PROGRAM Alarm_conv_3
VAR
bAlarm_b3_S1_SB0_blink	:BOOL;
bAlarm_b3_S6_SB0_blink	:BOOL;
END_VAR

//Нет готовности конвейер 3	
	bAlarm3QF2_3QF7 S=NOT b_3QF2_3QF7 	AND bPermAlarm1;
	bAlarm3QF8 		S=NOT b_3QF8 		AND bPermAlarm1;
//	bAlarm3KM2 		S=NOT b_3KM2 		AND bPermAlarm1;
//	bAlarm3KM3 		S=NOT b_3KM3 		AND bPermAlarm1;
//	bAlarm3KM4 		S=NOT b_3KM4 		AND bPermAlarm1;
//	bAlarm3KM5 		S=NOT b_3KM5 		AND bPermAlarm1;
//	bAlarm3KM6 		S=NOT b_3KM6 		AND bPermAlarm1;
//	bAlarm3KM7 		S=NOT b_3KM7 		AND bPermAlarm1;
	
//Грибки
	bAlarm_b3_S1_SB0 S=NOT   b3_S1_SB0 	AND bPermAlarm1;
	bAlarm_b3_S6_SB0 S=NOT   b3_S6_SB0 	AND bPermAlarm1;

// Индикация на грибках
	b3S1_SB0 := NOT b3_S1_SB0 AND blink.OUT;
	b3S6_SB0 := NOT b3_S6_SB0 AND blink.OUT;	
	
	blink(ENABLE:=bAlarm_b3_S1_SB0,TIMELOW:=T#500MS,TIMEHIGH:=T#500MS);
	bAlarm_b3_S1_SB0_blink := blink.OUT AND bAlarm_b3_S1_SB0;
	bAlarm_b3_S6_SB0_blink := blink.OUT AND bAlarm_b3_S6_SB0;	
(*Авария безопасности*)
	bAlarmSafety3 := bAlarm_b3_S1_SB0 OR bAlarm_b3_S6_SB0;

(*Нет общей готовности конвейера 1*)
	bNotReady_3 := bAlarm3QF2_3QF7 OR bAlarm3QF8 OR bAlarm3KM2 OR bAlarm3KM3 OR bAlarm3KM4 OR bAlarm3KM5 OR bAlarm3KM6 OR bAlarm3KM7;
					
IF  bNotReady3 THEN  sAlarm3:="Нет готовности 3";
		ELSIF bAlarmSafety3 THEN  sAlarm2:="Авария безопасности 3";
			ELSE sAlarm3:="---------";
END_IF

	bPermAlarmDrive3 := bPermAlarm1 AND NOT bAlarmSafety3;

(*(*Готовность *)
	IF NOT bDriveReady3s01M1 AND bPermAlarmDrive3  THEN  bNotDriveReady3s01M1 := TRUE;
	END_IF    
	IF NOT bDriveReady3s02M1 AND bPermAlarmDrive3  THEN  bNotDriveReady3s02M1 := TRUE;
	END_IF 
	IF NOT bDriveReady3s03M1 AND bPermAlarmDrive3  THEN  bNotDriveReady3s03M1 := TRUE;
	END_IF 
	IF NOT bDriveReady3s04M1 AND bPermAlarmDrive3  THEN  bNotDriveReady3s04M1 := TRUE;
	END_IF 
	IF NOT bDriveReady3s05M1 AND bPermAlarmDrive3  THEN  bNotDriveReady3s05M1 := TRUE;
	END_IF 
	IF NOT bDriveReady3s06M1 AND bPermAlarmDrive3  THEN  bNotDriveReady3s06M1 := TRUE;
	END_IF*)

(*Долгие перемещения Drive*)
	IF bLongMove3s01_s02_1   THEN bLongMove_3s01_s02_1 := TRUE;
	END_IF
	IF bLongMove3s02_1_s02_2  THEN bLongMove_3s02_1_s02_2 := TRUE;
	END_IF
	IF bLongMove3s02_2_s03_1  THEN bLongMove_3s02_2_s03_1 := TRUE;
	END_IF
	IF bLongMove3s02_s03  THEN bLongMove_3s02_s03 := TRUE;
	END_IF
		IF bLongMove3s03_1_s03_2   THEN bLongMove_3s03_1_s03_2 := TRUE;
	END_IF
	IF bLongMove3s03_2_s04_1  THEN bLongMove_3s03_2_s04_1 := TRUE;
	END_IF
	IF bLongMove3s03_s04  THEN bLongMove_3s03_s04 := TRUE;
	END_IF
	IF bLongMove3s04_1_s04_2  THEN bLongMove_3s04_1_s04_2 := TRUE;
	END_IF
		IF bLongMove3s04_2_s05   THEN bLongMove_3s04_2_s05  := TRUE;
	END_IF
	IF bLongMove3s05_1s06  THEN bLongMove_3s05_1s06 := TRUE;	
	END_IF
	
(*Нет готовности*)
	bNotReady3 := bNotDriveReady3s01M1 OR bNotDriveReady3s02M1 OR bNotDriveReady3s03M1 OR
			  bNotDriveReady3s04M1 OR bNotDriveReady3s05M1 OR bNotDriveReady3s06M1;

(*Долгое премещение*)
	bLongMove3 :=bLongMove_3s02_1_s02_2 OR bLongMove_3s02_1_s02_2  OR bLongMove_3s02_s03 OR
	       bLongMove_3s03_1_s03_2 OR bLongMove_3s03_2_s04_1 OR bLongMove_3s03_s04 OR bLongMove_3s04_1_s04_2 OR
			bLongMove_3s04_2_s05   OR bLongMove_3s05_1s06;


(*Сброс бита аварии по кнопке с панели*)
	bAlarmReset3 := bButtAlarmReset3;

(*Восстановление/сброс аварийных сигналов*)
IF bReset3 OR bAlarmReset3 THEN
	bAlarm3QF8 :=FALSE; bAlarm3QF2_3QF7 :=FALSE; 
	bAlarm3KM2 :=FALSE; bAlarm3KM3 :=FALSE; bAlarm3KM4 :=FALSE; bAlarm3KM5 :=FALSE; bAlarm3KM6 :=FALSE; bAlarm3KM7 :=FALSE;

	bNotDriveReady3s01M1 := FALSE; bNotDriveReady3s02M1 := FALSE; bNotDriveReady3s03M1 := FALSE;
	bNotDriveReady3s04M1 := FALSE; bNotDriveReady3s05M1 := FALSE; bNotDriveReady3s06M1 := FALSE;
	
	bLongMove_3s02_1_s02_2 := FALSE;bLongMove_3s02_1_s02_2 := FALSE; bLongMove_3s02_s03 := FALSE;
	bLongMove_3s03_1_s03_2 := FALSE; bLongMove_3s03_2_s04_1:= FALSE; bLongMove_3s03_s04 := FALSE;
	 bLongMove_3s04_1_s04_2:= FALSE;  bLongMove_3s04_2_s05 := FALSE;
    bLongMove_3s05_1s06 := FALSE;
	
	
	bAlarm_b3_S1_SB0 := FALSE; bAlarm_b3_S6_SB0 := FALSE;
END_IF

(*Формирование аварии*)
	bAlarm3 := bNotReady3 OR bLongMove3 OR bAlarmSafety3 OR bNotReady_3 OR bNotReadyGeneral OR bOverflow_CTU_Weight3 OR bOverflow_CTU_ID3;
	bAlarm3_vis := blink.OUT AND bAlarm3;
	
IF  bNotReady3 THEN  sAlarmLine3:="Нет готовности 3";
		ELSIF bLongMove3 THEN   sAlarmLine3:="Долгое перемещение 3";
			ELSE sAlarmLine3:="---------";
END_IF
IF bAlarm3 AND b_3AS1 THEN bRed_3S1HL1 :=TRUE; bRed_3S1_HL1 := TRUE;
	ELSE bRed_3S1HL1 := FALSE; bRed_3S1_HL1 := FALSE;
END_IF
AlarmEvent_conv3();

END_PROGRAM

(* stored: Version 1.1.0.1, ProductVersion 3.1.4024.4
   POU Alarm_conv_3: Id {5f708db7-1076-41b8-bcdb-e6a421b382fb}, SpecialFunc None *)
